// TIA Portal V20 export
TYPE "typeCmControlNode"
// stored: Namespace Unit1.Em3
   STRUCT
      interlock : "Unit1.Em3.typeCmControlNodeInterlock";
      command : "Unit1.Em3.typeCmControlNodeCommand";
      softcam : "Unit1.Em3.typeCmControlNodeSoftCam";
   END_STRUCT;
END_TYPE
